FUNCTION_BLOCK ReferenceBlock

VAR
	stStopStatus	:ST_StopStatus;
	refStopStatus	:REFERENCE TO ST_StopStatus;
END_VAR

refStopStatus REF= stStopStatus;

END_FUNCTION_BLOCK

(* stored: Version 1.1.0.1, ProductVersion 3.1.4024.10
   POU ReferenceBlock: Id {48b98226-5d65-43d8-a488-486dd48bd879}, SpecialFunc None *)
